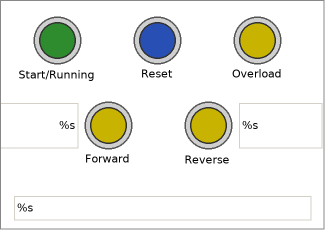
VISUALIZATION V_MC  // 325x230
    Lamp1 (30,13 55x55), variable: Module_IO.oStartLamp, style: Lamp-Lamp1-Green
    Label (9,60 95x30), "Start/Running"
    Lamp1 (130,13 55x55), variable: Module_IO.oResetButton, style: Lamp-Lamp1-Blue
    Label (108,59 98x30), "Reset"
    Lamp1 (81,98 55x55), variable: Module_IO.oForward, style: Lamp-Lamp1-Yellow
    Lamp1 (181,98 55x55), variable: Module_IO.oReverse, style: Lamp-Lamp1-Yellow
    Label (64,144 87x30), "Forward"
    Label (166,145 82x30), "Reverse"
    Textfield (14,196 297x24), "%s", text variable: MC.sState
    Textfield (0,103 78x45), "%s", text variable: MC.tForward, invisible if: NOT (Module_IO.iForward AND MC.bTimerOff)
    Textfield (239,103 83x45), "%s", text variable: MC.tReversing, invisible if: NOT (Module_IO.iReverse AND MC.bTimerOff)
    Lamp1 (230,13 55x55), variable: Module_IO.iMotorOverLoad, style: Lamp-Lamp1-Yellow
    Label (208,59 98x30), "Overload"
END_VISUALIZATION

(* stored: Version 1.1.0.1, ProductVersion 3.1.4024.11
   Visu V_MC: Id {00283fe0-240d-4bed-8557-b198c847978c} *)
